INTERFACE I_AnalogInput EXTENDS I_Channel

PROPERTY P_Value : LREAL
GET
END_GET
END_PROPERTY

END_INTERFACE

(* stored: Version 1.1.0.1
   Itf I_AnalogInput: Id {99b1c711-8580-0ac0-2f30-4876ffd850f4}
   Property P_Value: Id {49551ec9-ec98-03d6-0acc-454beece07a8}
   Get Get: Id {62963b61-2744-02cc-298a-1b68e57dc146} *)
